PROGRAM MAIN
VAR
END_VAR

END_PROGRAM

(* stored: Version 1.1.0.1
   POU MAIN: Id {831f0fe4-bb3b-41e1-96ac-a133bf163627}, SpecialFunc None *)
